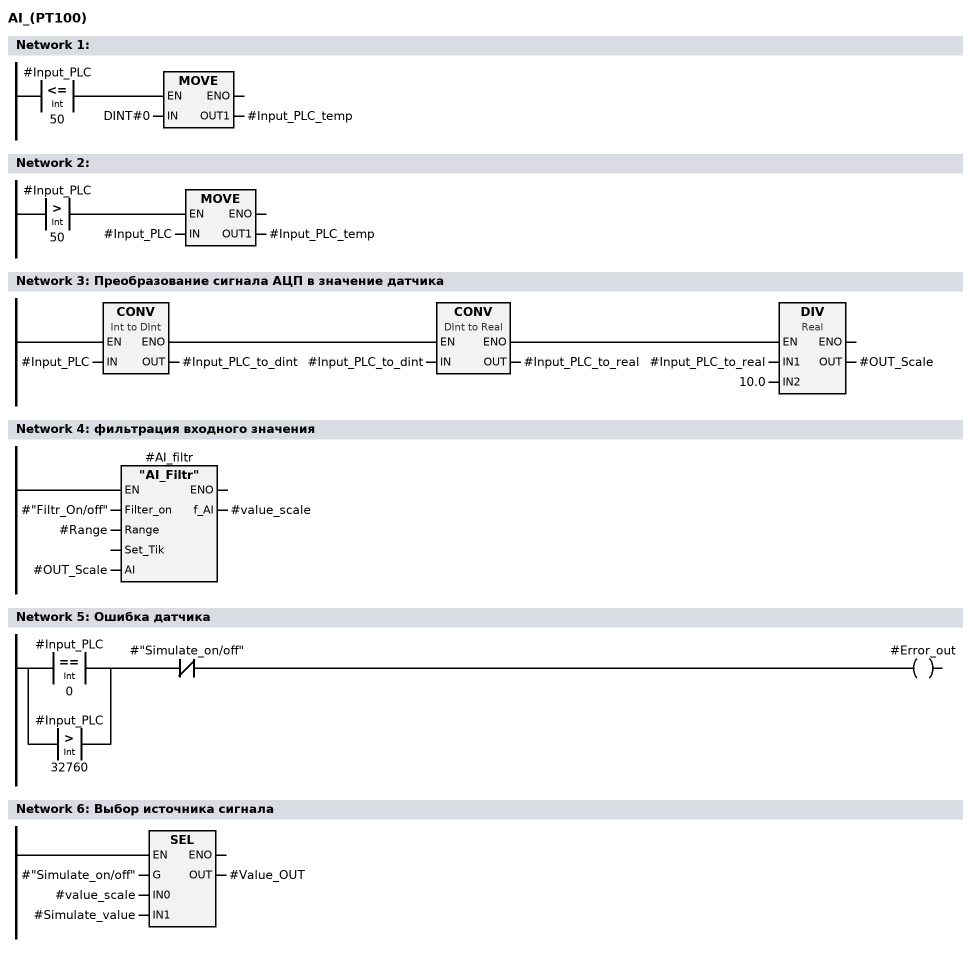
   RUNG wire#powerrail
      { S7_Templates := "SrcType := Int" } LE_Contact(in1 := #Input_PLC, in2 := 50)
      { S7_GenerateENO := "TRUE" } Move(in := DINT#0, out1 => #Input_PLC_temp)
   END_RUNG
   // the same network as SCL:
   IF #Input_PLC <= 50 THEN #Input_PLC_temp := DINT#0; END_IF;
END_REGION

REGION Network 2
   RUNG wire#powerrail
      { S7_Templates := "SrcType := Int" } GT_Contact(in1 := #Input_PLC, in2 := 50)
      { S7_GenerateENO := "TRUE" } Move(in := #Input_PLC, out1 => #Input_PLC_temp)
   END_RUNG
   // the same network as SCL:
   IF #Input_PLC > 50 THEN #Input_PLC_temp := #Input_PLC; END_IF;
END_REGION

REGION Network 3: Преобразование сигнала АЦП в значение датчика
   RUNG wire#powerrail
      { S7_Templates := "[SrcType := Int, DestType := DInt]"; S7_GenerateENO := "TRUE" } Convert(in := #Input_PLC, out => #Input_PLC_to_dint)
      { S7_Templates := "[SrcType := DInt, DestType := Real]"; S7_GenerateENO := "TRUE" } Convert(in := #Input_PLC_to_dint, out => #Input_PLC_to_real)
      { S7_Templates := "SrcType := Real"; S7_GenerateENO := "TRUE" } Div(in1 := #Input_PLC_to_real, in2 := 10.0, out => #OUT_Scale)
   END_RUNG
   // the same network as SCL:
   // ENO of a box is taken as its EN; it also drops when the box reports an error
   #Input_PLC_to_dint := INT_TO_DINT(#Input_PLC);
   #Input_PLC_to_real := DINT_TO_REAL(#Input_PLC_to_dint);
   #OUT_Scale := #Input_PLC_to_real / 10.0;
END_REGION

REGION Network 4: фильтрация входного значения
   RUNG wire#powerrail
      #AI_filtr(Filter_on := #"Filtr_On/off", Range := #Range, Set_Tik :=, AI := #OUT_Scale, f_AI => #value_scale)
   END_RUNG
   // the same network as SCL:
   #AI_filtr(Filter_on := #"Filtr_On/off", Range := #Range, AI := #OUT_Scale, f_AI => #value_scale);   // "AI_Filtr"
END_REGION

REGION Network 5: Ошибка датчика
   RUNG wire#powerrail
      { S7_Templates := "SrcType := Int" } EQ_Contact(in1 := #Input_PLC, in2 := 0)
      wire#w1
      I_Contact( #"Simulate_on/off" )
      Coil( #Error_out )
   END_RUNG
   RUNG wire#powerrail
      { S7_Templates := "SrcType := Int" } GT_Contact(in1 := #Input_PLC, in2 := 32760)
   END_RUNG wire#w1
   // the same network as SCL:
   #Error_out := ((#Input_PLC = 0) OR (#Input_PLC > 32760)) AND NOT #"Simulate_on/off";
END_REGION

REGION Network 6: Выбор источника сигнала
   #Value_OUT := SEL(G := #"Simulate_on/off", IN0 := #value_scale, IN1 := #Simulate_value);
END_REGION
END_FUNCTION_BLOCK

// folder: AI_Signal/Funktion

FUNCTION_BLOCK "AI_Filtr"   // FB14, SCL
{ S7_Optimized_Access := 'FALSE' }
VERSION : 0.1
   VAR_INPUT
      Filter_on : Bool;   // Вкл фильтрации
      Range : Int := 10;   // Кол-во входных значений для вычисления среднего
      Set_Tik : Int := 2;   // Задача периода фильтрации от 1(мин) до 8
      AI : Real;   // Вход значения датчика
   END_VAR
   VAR_OUTPUT
      f_AI : Real;   // выход значения с фильтром или без
   END_VAR
   VAR
      CTU : CTU_INT;   // счетчик для подсчета кол-во вх значений
      Tik : Bool;   // Время фильтрации
      ai_array : Array[0..#Max_Array] of Real;   // Массив значений датчика
      i : Int;   // для цикла ФОР
      sum_AI : Real;   // Суммирование значений с входа датчика
      Avarage_AI : Real;   // Среднее значение датчика
      fRS_set : Bool;   // Для RS тригера
      fRS_res : Bool;   // Для RS тригера
      fRS_out : Bool;   // Для RS тригера
      FullFiltr : Bool;   // Ожидание наполнения значений для вычисления средней
      Res_count : Bool;   // сброс счетчика
   END_VAR
   VAR CONSTANT
      Max_Array : Int := 30;   // Размер массива
   END_VAR
BEGIN

   CASE #Set_Tik OF                   
       1:  
           #Tik := "Time_0.1s";
       2:  
           #Tik := "Time_0.2s";
       3:
           #Tik := "Time_0.4s";
       4:
           #Tik := "Time_0.5s";
       5:
           #Tik := "Time_0.8s";
       6:
           #Tik := "Time_1s";
       7:
           #Tik := "Time_1.6s";
       8:
           #Tik := "Time_2s";
       0:
           #Tik := "Time_0.1s";

       ELSE  
           #Set_Tik := 8;
   END_CASE;  // Выбор периода фильтрации входного сигнала
   REGION RS триггер
       IF #fRS_set THEN
           #fRS_out := true;
       ELSIF #fRS_res AND NOT #fRS_set THEN
           #fRS_out := false;
       END_IF;
   END_REGION

   REGION Подсчет среднего значения входа
       // Statement section REGION
           #CTU(CU := #Tik,
                PV := #Range,
                R := #Res_count,
                Q => #Res_count);                                      // Счетчик для набора значений с входа
           #ai_array[#CTU.CV] := #AI;                                  // Запись значений с входа в массив

           IF #Res_count THEN                                              // СБРОС как счетчик переполниться Для корректной работы счетчика
               #i := 0;
               #sum_AI := 0;
           END_IF;

           IF #Range <> #i THEN                                    // выход из цикла FOR при суммировании всех значений, почему то сам не прекращел подсчет при окончании цикла все время суммировался 
               FOR #i := 0 TO (#Range - 1) DO
                   #sum_AI := #ai_array[#i] + #sum_AI;             // суммирование значений
               END_FOR;
           END_IF;

       #Avarage_AI := #sum_AI / #Range;                             // Вычисление среднего значения
       #fRS_res := NOT #Filter_on;

   END_REGION

   REGION Выбор выхода прямое или фильтрованное значение
       IF #Filter_on THEN                                          //Включение выключение фильтрации
           #fRS_set := #CTU.QD;                                    //При включении фильтра ждем наполнения значениями с входа, пока ждем - отправляем на выход прямое значение входа, далее фильтруем
            #FullFiltr := #fRS_out;

          IF #FullFiltr THEN                                       //Когда фильтр наполнился - вывыодим среднее значение входа
               #f_AI := #Avarage_AI;                              // ЗАпись значения на выход AI
          ELSE
               #f_AI := #AI;                                     // Прямой вывод значения, пока значения не наполнились данными
          END_IF;
       ELSE
           #f_AI := #AI;                                        // Если фильтр выключен, на выход прямое значение с входа
       END_IF; 

   END_REGION
END_FUNCTION_BLOCK

FUNCTION "Calculate_AI" : Void   // FC7, SCL
{ S7_Optimized_Access := 'FALSE' }
VERSION : 0.1
   VAR_INPUT
      IN_sensors : Int;
      Current_max : Real;
      Current_min : Real;
      Code_HL : Real;
      Code_LL : Real;
      Param_Sensor_HL : Real;   // Параметры датчика по паспорту (макс значение)bar, C, итд
      Param_Sensor_LL : Real;   // Параметры датчика по паспорту (мин значение)bar, C, итд
   END_VAR
   VAR_OUTPUT
      signal_Electric : Real;   // выход в электрических ед измерения
      Value_Sensor : Real;   // выход реального значения датчика в ед измерения
   END_VAR
   VAR_TEMP
      sensor_to_real : Real;   // Для конвертации INT to Real
      result_to_out_signal : Real;   // Для вычитания реального значения показания датчика
   END_VAR
BEGIN
       //Convert int to real
   #sensor_to_real := INT_TO_REAL(#IN_sensors);

       // Расчет значения АЦП контроллера в значение эл. ед измерения (I, U) в зависимости от значений на входе
   #signal_Electric := ((#sensor_to_real - #Code_LL) * (#Current_max - #Current_min) / (#Code_HL - #Code_LL))+ #Current_min;
   #result_to_out_signal := #signal_Electric;

   // Расчет значения в реальных единицах измерения датчика (bar, C,) в зависимости от введеных параметров датчика Param_Sensor min/max
   #Value_Sensor := (#result_to_out_signal - #Current_min) * (#Param_Sensor_HL - #Param_Sensor_LL) / (#Current_max - #Current_min) + #Param_Sensor_LL;
END_FUNCTION

// folder: DI_signal

FUNCTION_BLOCK "FB_DI"   // FB15, LAD
TITLE = Блок обработки дискретных входов
{ S7_Optimized_Access := 'FALSE' }
VERSION : 0.1
   VAR_INPUT
      input_value : Bool;   // Входной тэг контроллера
   END_VAR
   VAR_OUTPUT
      Value : Bool;   // Обработанный сигнал
   END_VAR
   VAR_IN_OUT
      stParamDI : "Tipe_DI";
   END_VAR
   VAR
      Time_Delay : Time;   // Время фильтрации для таймера
      Time_On : TON_TIME;   // Фильтр на Вкл
      Time_Off : TON_TIME;   // Фильтр на Выкл
      Nul_Time : Time := T#1MS;   // Откл фильтрации (0)
      bOut_Value : Bool;
   END_VAR
BEGIN

REGION Network 1: Включение фильтрации
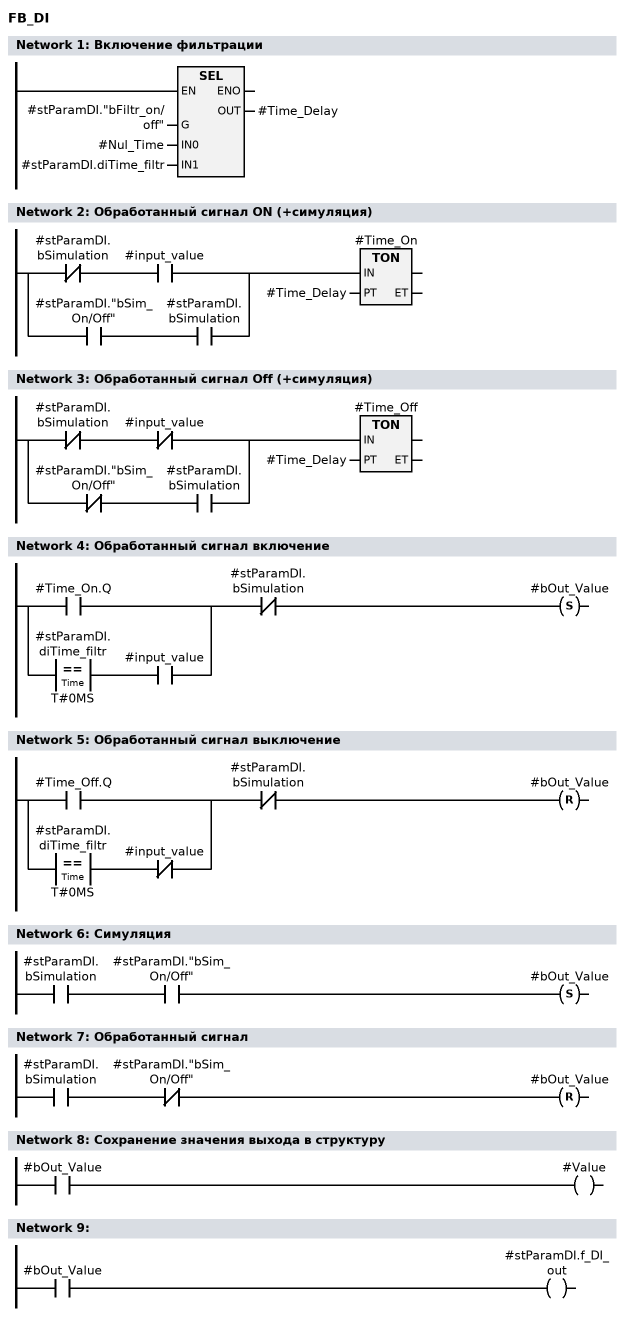
   #Time_Delay := SEL(G := #stParamDI."bFiltr_on/off", IN0 := #Nul_Time, IN1 := #stParamDI.diTime_filtr);
END_REGION

REGION Network 2: Обработанный сигнал ON (+симуляция)
   #Time_On(IN := (NOT #stParamDI.bSimulation AND #input_value) OR (#stParamDI."bSim_On/Off" AND #stParamDI.bSimulation),   // TON
            PT := #Time_Delay);
END_REGION

REGION Network 3: Обработанный сигнал Off (+симуляция)
   #Time_Off(IN := (NOT #stParamDI.bSimulation AND NOT #input_value) OR (NOT #stParamDI."bSim_On/Off" AND #stParamDI.bSimulation),   // TON
             PT := #Time_Delay);
END_REGION

REGION Network 4: Обработанный сигнал включение
   RUNG wire#powerrail
      Contact( #Time_On.Q )
      wire#w1
      I_Contact( #stParamDI.bSimulation )
      S_Coil( #bOut_Value )
   END_RUNG
   RUNG wire#powerrail
      { S7_Templates := "SrcType := Time" } EQ_Contact(in1 := #stParamDI.diTime_filtr, in2 := T#0MS)
      Contact( #input_value )
   END_RUNG wire#w1
   // the same network as SCL:
   IF (#Time_On.Q OR ((#stParamDI.diTime_filtr = T#0MS) AND #input_value)) AND NOT #stParamDI.bSimulation THEN
       #bOut_Value := TRUE;
   END_IF;
END_REGION

REGION Network 5: Обработанный сигнал выключение
   RUNG wire#powerrail
      Contact( #Time_Off.Q )
      wire#w1
      I_Contact( #stParamDI.bSimulation )
      R_Coil( #bOut_Value )
   END_RUNG
   RUNG wire#powerrail
      { S7_Templates := "SrcType := Time" } EQ_Contact(in1 := #stParamDI.diTime_filtr, in2 := T#0MS)
      I_Contact( #input_value )
   END_RUNG wire#w1
   // the same network as SCL:
   IF (#Time_Off.Q OR ((#stParamDI.diTime_filtr = T#0MS) AND NOT #input_value)) AND NOT #stParamDI.bSimulation THEN
       #bOut_Value := FALSE;
   END_IF;
END_REGION

REGION Network 6: Симуляция
   RUNG wire#powerrail
      Contact( #stParamDI.bSimulation )
      Contact( #stParamDI."bSim_On/Off" )
      S_Coil( #bOut_Value )
   END_RUNG
   // the same network as SCL:
   IF #stParamDI.bSimulation AND #stParamDI."bSim_On/Off" THEN #bOut_Value := TRUE; END_IF;
END_REGION

REGION Network 7: Обработанный сигнал
   RUNG wire#powerrail
      Contact( #stParamDI.bSimulation )
      I_Contact( #stParamDI."bSim_On/Off" )
      R_Coil( #bOut_Value )
   END_RUNG
   // the same network as SCL:
   IF #stParamDI.bSimulation AND NOT #stParamDI."bSim_On/Off" THEN #bOut_Value := FALSE; END_IF;
END_REGION

REGION Network 8: Сохранение значения выхода в структуру
   RUNG wire#powerrail
      Contact( #bOut_Value )
      Coil( #Value )
   END_RUNG
   // the same network as SCL:
   #Value := #bOut_Value;
END_REGION

REGION Network 9
   RUNG wire#powerrail
      Contact( #bOut_Value )
      Coil( #stParamDI.f_DI_out )
   END_RUNG
   // the same network as SCL:
   #stParamDI.f_DI_out := #bOut_Value;
END_REGION
END_FUNCTION_BLOCK

// folder: FB - All

FUNCTION_BLOCK "R_trig"   // FB16, SCL
{ S7_Optimized_Access := 'TRUE' }
VERSION : 0.1
   VAR_INPUT
      In : Bool;
   END_VAR
   VAR_OUTPUT
      Q : Bool;
   END_VAR
   VAR
      Click_M : Bool;
   END_VAR
BEGIN
   #Q := #In AND NOT #Click_M;
   #Click_M := #In;
END_FUNCTION_BLOCK

// folder: FB - All/LogickBlocks

FUNCTION_BLOCK "Pump"   // FB1, SCL
{ S7_Optimized_Access := 'FALSE' }
VERSION : 0.1
   VAR_INPUT
      bManualMode : Bool;   // Выбор ручного режима
      bManualStart : Bool;   // Ручной режим - старт
      bManualStop : Bool;   // Ручной режим - стоп
      rManualSpeed : Real;   // Ручной режим - скорость
      bDryRunn : Bool;   // Защита от сухого хода
      bAutoSTop : Bool;   // Остановка насоса
      bAutoStartPerm : Bool;   // Команда на работоу в авто режиме
      rAutoSpeed : Real;   // Скорость в авто режиме
      bАвтоматы : Bool;   // Готовность привода (автоматы)
      bПускатели : Bool;   // Готовность Пускателя
      bDriveRunning : Bool;   // Привод в работе
      bDriveFault : Bool;   // Привод в ошибке
      rMinSpeed : Real;   // Минимальная скорость
      rMaxSpeed : Real := 100.0;   // Максимальная скорость
      bResetFault : Bool;   // Сброс аварии
   END_VAR
   VAR_OUTPUT
      bRunCmd : Bool;   // Пуск частотника
      iSpeedOut : Int;   // Скорость насоса для аналогового выхода
      "rSpeedHMI(0-100)" : Real;   // Скорость работы (0-100) для HMI
      bPumpRunning : Bool;   // Работа
      bPumpFault : Bool;   // Авария
      iStatus : Int;   // Статус (0 - стоп 1 - работа 2 - авария)
   END_VAR
   VAR
      bFaultLatch : Bool;
      bRunRequest : Bool;
      rSpeedPump : Real;   // Скорость насоса
      TON_NotStartRun : TON_TIME;   // ТАймер ожидания сигнала о запуске
      TON_NotContactRun : TON_TIME;   // ТАймер ожидания с контактора
      TON_DryRun : TON_TIME;   // Таймер сухого хода
   END_VAR
BEGIN
   (*
   // 1. Обработка аварий
   // Обработка ожидания сигнала о работе после старта
   IF #bAutoStartPerm THEN
       ;

   END_IF;
   *)

   // 1 Ручной режим
   IF #bManualMode THEN
       // Ручной режим
       IF #bManualStart AND NOT #bManualStop THEN
           #bRunRequest := TRUE;
       ELSIF #bManualStop THEN // OR NOT #bАвтоматы THEN
           #bRunRequest := FALSE;
       END_IF;
   ELSE
       // Автоматический режим
       // 
       //Обработка аварий
       //
       //Таймер ожидания останова по сухому ходу
       #TON_DryRun(IN := NOT #bDryRunn,
                   PT := t#1s);    //
       //--------------------------------------------------------------------------------------------------------
       IF #bAutoStartPerm AND NOT #bAutoSTop AND #bDryRunn THEN
           #TON_NotStartRun(IN := NOT #bDriveRunning AND #bDryRunn, PT := t#5s);  //Таймер ожидания сигнала подтверждения пуска от частотника
           #TON_NotContactRun(IN := NOT #bПускатели, PT := t#10s);  //Таймер ожидания сигнала подтверждения пуска от пускателя


       ELSE
           #TON_NotStartRun(IN :=FALSE,PT := t#5s);
           #TON_NotContactRun(IN := FALSE,PT := t#5s);
       END_IF;
       #bFaultLatch := #TON_NotStartRun.Q OR #TON_NotContactRun.Q OR (#bDriveFault OR NOT #bАвтоматы) OR (NOT #bResetFault AND #bFaultLatch); //Разкоментировать если нужна будет фиксация АЛАРМА, сброс только по входу РЕСЕТ
       #bPumpFault := #bFaultLatch;

       //Старт--------------------------------
       #bRunRequest := #bAutoStartPerm AND NOT #bPumpFault AND NOT #TON_DryRun.Q;
   END_IF;

   // 3. Задание скорости
   IF #bManualMode THEN
       #"rSpeedHMI(0-100)" := LIMIT(MN := #rMinSpeed, IN := #rManualSpeed, MX := #rMaxSpeed);
   ELSE
       #"rSpeedHMI(0-100)" := LIMIT(MN := #rMinSpeed, IN := #rAutoSpeed, MX := #rMaxSpeed);
   END_IF;

   // Преобразование значения от 0-100 до 0-27648 для аналогового выхода
   #iSpeedOut := REAL_TO_INT((#"rSpeedHMI(0-100)"/ 100.0) * 27648.0);

   // 4. Выходные команды и статусы
   // Команды старт
   #bRunCmd := #bRunRequest;

   //Выход статуса для HMI
   #bPumpRunning := #bDriveRunning AND #bRunCmd AND NOT #bAutoSTop OR (#bManualStart AND #bManualMode);



   // 5. Числовой статус (для HMI/SCADA)
   IF #bFaultLatch THEN
       #iStatus := 2; // Авария
   ELSIF #bPumpRunning THEN
       #iStatus := 1; // Работа
   ELSE
       #iStatus := 0; // Стоп
   END_IF;

   IF #bAutoSTop AND NOT #bManualMode THEN
       #bRunCmd := FALSE;
   END_IF;
END_FUNCTION_BLOCK

FUNCTION_BLOCK "FB_GlobalStateManager"   // FB2, SCL
{ S7_Optimized_Access := 'FALSE' }
VERSION : 0.1
   VAR_INPUT
      bStartCmd : Bool;   // Команда на старт от HMI
      bConfirmStart : Bool;   // Подтверждение оператора
      bResetFault : Bool;   // Сброс ошибки
      bAllSetpointsReached : Bool;   // // Все температуры достигли уставок
      bNoFaults : Bool;   // Нет аварий
      tStartTimeout : Time := T#30m;   // Время за которое пастер выходит на режим
      tReadyDelay : Time := t#10s;   // Время ожидания при выходе на режим до готовности
   END_VAR
   VAR_OUTPUT
      eState : Int;   // Текущее состояние
      bConveyorEnable : Bool;   // Разрешение на работу конвейера
      bSystemReady : Bool;   // Готовность системы
      bSystemFault : Bool;   // Состояние Fault
      sStatusText : WString;   // Текст для HMI
   END_VAR
   VAR
      tonStartTimeout : TON_TIME;   // Таймер выхода на режим
      tonReadyDelay : TON_TIME;   // Таймер готовности
   END_VAR
   VAR CONSTANT
      cSTATE_IDLE : Int;
      cSTATE_CHECK : Int := 10;
      cSTATE_STARTING : Int := 20;
      cSTATE_READY_DELAY : Int := 30;
      cSTATE_READY : Int := 40;
      cSTATE_FAULT : Int := 99;
      sText1 : String := 'Waiting';
   END_VAR
BEGIN
   // Сброс таймеров при неактивных состояниях (по требованию 1)
   IF #eState <> #cSTATE_STARTING THEN
       #tonStartTimeout(IN := FALSE,
                        PT := #tStartTimeout);
   END_IF;

   IF #eState <> #cSTATE_READY_DELAY THEN
       #tonReadyDelay(IN := FALSE,
                      PT := #tReadyDelay);
   END_IF;

   // Глобальная проверка аварии (по требованию 4)
   IF NOT #bNoFaults AND #eState <> #cSTATE_FAULT THEN
       #eState := #cSTATE_FAULT;
       #bSystemFault := TRUE;
       #bConveyorEnable := FALSE; // Принудительный останов (по требованию 2)
   ELSIF NOT #bStartCmd THEN
       #eState := #cSTATE_IDLE;
   END_IF;


   REGION Основная логика

       // Основной CASE
       CASE #eState OF
           #cSTATE_IDLE:
               #bConveyorEnable := FALSE;
               IF #bStartCmd AND #bNoFaults THEN // Запрет старта при аварии
                   #eState := #cSTATE_CHECK;
               END_IF;

           #cSTATE_CHECK:
               // Проверка уже в глобальном условии, дублирование не нужно
               #eState := #cSTATE_STARTING;

           #cSTATE_STARTING:
               IF #bAllSetpointsReached THEN
                   #eState := #cSTATE_READY_DELAY;
               ELSIF #tonStartTimeout.Q THEN
                   #eState := #cSTATE_FAULT;
               END_IF;

           #cSTATE_READY_DELAY:
               IF #tonReadyDelay.Q THEN
                   #eState := #cSTATE_READY;
               END_IF;

           #cSTATE_READY:
               #bSystemReady := TRUE;
               IF #bConfirmStart THEN
                   #bConveyorEnable := TRUE;
               END_IF;

           #cSTATE_FAULT:
               #bSystemFault := TRUE;
               #bConveyorEnable := FALSE; // Гарантированный останов
               IF #bResetFault AND #bNoFaults THEN
                   #eState := #cSTATE_IDLE;
                   #bSystemFault := FALSE;
               END_IF;

           ELSE
               #eState := #cSTATE_IDLE;
       END_CASE;

   END_REGION


   // Обновление таймеров (после логики состояний!)
   #tonStartTimeout(IN := (#eState = #cSTATE_STARTING) AND NOT #bAllSetpointsReached,
                    PT := #tStartTimeout);
   #tonReadyDelay(IN := (#eState = #cSTATE_READY_DELAY),
                  PT := #tReadyDelay);
END_FUNCTION_BLOCK

FUNCTION_BLOCK "Valve(c/o)"   // FB3, SCL
{ S7_Optimized_Access := 'FALSE' }
VERSION : 0.1
   VAR_INPUT
      bAuto_OpenCmd : Bool;   // Команда открыть (автомат)
      bManualMode : Bool;   // Ручной режим (TRUE)
      bManualOpen : Bool;   // Команда открыть в ручном режиме
      bFeedbackOpen : Bool;   // Обратная связь "Открыт"
      tMaxTime : Time;   // Время на открытие
      bResetAlarm : Bool;   // Сброс аварии
      bHaveFeedback : Bool;   // Есть ли обратная связь (0 - нет, 1 есть)
   END_VAR
   VAR_OUTPUT
      bValveOpen : Bool;   // Управляющий выход
      iValveState : Int;   // 0 = Закрыт, 1 = Открыт, 2 = Авария
      bValveFault : Bool;   // Авария
   END_VAR
   VAR
      tiOpenTimer : TON_TIME;   // Таймер на открытие
      bWaitingOpen : Bool;   // Флаг ожидания открытия
      bEnableTimer : Bool;   // Флаг активации таймера
   END_VAR
BEGIN

   // Обновление таймера — всегда в одном месте, вне условий
   #tiOpenTimer(
                IN := #bEnableTimer,
                PT := #tMaxTime
   );

   // Сброс
   IF #bResetAlarm THEN
       #bValveFault := FALSE;
       #bWaitingOpen := FALSE;
       #bEnableTimer := FALSE;
   END_IF;

   // === Режим: РУЧНОЙ ===
   IF #bManualMode THEN
       #bValveOpen := #bManualOpen;
       #bValveFault := FALSE;          // Аварии в ручном режиме не учитываются
       #bEnableTimer := FALSE;
       #bWaitingOpen := FALSE;

       // === Режим: АВТО ===
   ELSE

           // Управление выходом с учетом аварии, с контролем обратной связи
        IF #bAuto_OpenCmd AND NOT #bValveFault THEN
                   #bValveOpen := TRUE;
        ELSE
                   #bValveOpen := FALSE;
               END_IF;

               //  Проверяем, есть ли контроль обратной связи
        IF #bHaveFeedback THEN
            // Контроль открытия
            IF #bAuto_OpenCmd AND NOT #bFeedbackOpen AND NOT #bValveFault THEN
                #bEnableTimer := TRUE;
                #bWaitingOpen := TRUE;
            ELSE
                #bEnableTimer := FALSE;
                ;
                IF #bFeedbackOpen THEN
                    #bWaitingOpen := FALSE;
                END_IF;
            END_IF;
        END_IF;


           // Авария
           IF #tiOpenTimer.Q AND #bWaitingOpen THEN
               #bValveFault := TRUE;
               #bWaitingOpen := FALSE;
           END_IF;

   END_IF;


   // Состояние клапана
   IF #bValveFault THEN
       #iValveState := 2;       // Авария
   ELSIF #bHaveFeedback AND #bFeedbackOpen  THEN
       #iValveState := 1;       // Открыт
   ELSIF NOT #bHaveFeedback AND (NOT #bManualMode AND #bAuto_OpenCmd) OR (#bManualOpen AND #bManualMode) THEN
       #iValveState := 1;       // Открыт 
   ELSE
       #iValveState := 0;       // Закрыт
   END_IF;
END_FUNCTION_BLOCK

FUNCTION_BLOCK "Valve(regul)"   // FB4, SCL
{ S7_Optimized_Access := 'FALSE' }
VERSION : 0.1
   VAR_INPUT
      bManualMode : Bool;   // TRUE = ручной режим, FALSE = автоматический режим
      rAutoSetpoint : Real;   // Уставка открытия клапана в % (0.0–100.0) в автомате
      "bAutoOpen/Close" : Bool;   // Выход Do в автоматическом режиме
      rManualSetpoint : Real;   // Уставка открытия клапана в % (0.0–100.0) в ручном режиме
      "bManualOpen/Close" : Bool;   // Управление выходом открыть/закрыть
   END_VAR
   VAR_OUTPUT
      iAnalogOutput : Int;   // Значение для аналогового выхода (0–27648)
      rValvePosPercent : Real;   // Текущее % открытия клапана для HMI
      bStatusValveOpen : Int;   // Статус сигнал "клапан открыт" (TRUE, если >0%)
      "bOut_Open/Close" : Bool;   // выход для открытия клапана
   END_VAR
   VAR
      rSetpointPercent : Real;   // Расчётная уставка % открытия в текущем режиме
   END_VAR
BEGIN
       // Выбор уставки в зависимости от режима
       IF #bManualMode THEN
           #rSetpointPercent := #rManualSetpoint;
           #"bOut_Open/Close" := #"bManualOpen/Close";
       ELSE
           #rSetpointPercent := #rAutoSetpoint;
           #"bOut_Open/Close" := #"bAutoOpen/Close";
       END_IF;

       // Ограничение % от 0.0 до 100.0
       IF #rSetpointPercent < 0.0 THEN
           #rSetpointPercent := 0.0;
       ELSIF #rSetpointPercent > 100.0 THEN
           #rSetpointPercent := 100.0;
       END_IF;

       // Перевод % в значение для аналогового выхода
       #iAnalogOutput := REAL_TO_INT((#rSetpointPercent / 100.0) * 27648.0);

           // Вывод значения для HMI
       #rValvePosPercent := #rSetpointPercent;

       // Статус клапана для Панели HMI
       IF #rSetpointPercent > 0.0 AND #"bOut_Open/Close" THEN
           #bStatusValveOpen := 1;
       ELSE
           #bStatusValveOpen := 0;
       END_IF;
       ;
END_FUNCTION_BLOCK

FUNCTION_BLOCK "FB_Управление конвейером"   // FB5, SCL
{ S7_Optimized_Access := 'FALSE' }
VERSION : 0.1
   VAR_INPUT
      bEnable : Bool;   // Общий флаг работы системы
      bStartCmd : Bool;   // Команда на запуск от HMI, по кнопке из окна подтверждения
      bAllZonesInSetpoint : Bool;   // Все зоны достигли уставок
      bGlobalFault : Bool;   // Авария по системе
      bZoneHasPriority : Bool;   // У зоны с отклонением есть приоритет
      dwDeltaTempDelayMin : DWord;   // Задержка (мин), прежде чем остановить конвейер при отклонении
      dwResumeDelayMin : DInt;   // Время возврата после нормализации
   END_VAR
   VAR_OUTPUT
      bConveyorRun : Bool;   // Команда на пуск частотников
      bReadyToStart : Bool;   // Готовность к работе конвейера
      bWaitingConfirm : Bool;   // Ждём подтверждения от оператора, вывод окна на HMI
      bPaused : Bool;   // Конвейер остановлен по отклонению
   END_VAR
   VAR
      bStarted : Bool;   // Внутреннее состояние — процесс стартовал
      tiPauseTimer : TON_TIME;   // Таймер задержки перед остановкой
      tiResumeTimer : TON_TIME;   // Таймер ожидания перед возобновлением
      aZoneS_Status : Array[1..5] of "ZoneStatus";   // Массив для сбора состояния зон
      i : Int;
   END_VAR
   // tiPauseTimer.PT := T#1s;
   // tiResumeTimer.PT := T#1s;
BEGIN

   // Проверка на наличие флага обей работы системы
   IF NOT #bEnable THEN
       #bReadyToStart := FALSE;
       #bWaitingConfirm := FALSE;
       #bConveyorRun := FALSE;
       #bPaused := FALSE;
       #tiPauseTimer.IN := FALSE;
       #tiResumeTimer.IN := FALSE;
       RETURN;
   END_IF;



   // Условия готовности к запуску
   IF NOT #bStarted AND NOT #bGlobalFault AND #bAllZonesInSetpoint THEN
       #bReadyToStart := TRUE;

           // Команда на старт — вручную подтверждена
           IF NOT #bStartCmd THEN
               #bWaitingConfirm := TRUE;
           END_IF;

   ELSE
       #bReadyToStart := FALSE;
       #bWaitingConfirm := FALSE;
   END_IF;



   IF #bStartCmd AND #bReadyToStart THEN
       #bStarted := TRUE;
       #bWaitingConfirm := FALSE;
   END_IF;

   // После старта разрешаем работу, если нет аварий и температур в норме
   IF #bStarted AND NOT #bGlobalFault THEN

       IF NOT #bAllZonesInSetpoint THEN
           IF #bZoneHasPriority THEN
               // Включаем таймер паузы, задержка перед остановкой
               #tiPauseTimer(IN := TRUE,
                             PT := (#dwDeltaTempDelayMin * 60000)) //В минутах
               ;
           ELSE
               #tiPauseTimer(IN := FALSE,PT := t#0s);
           END_IF;

           // Переход в паузу
           IF #tiPauseTimer.Q THEN
               #bPaused := TRUE;
               #bConveyorRun := FALSE;
               #tiResumeTimer(IN := FALSE, PT := t#0s); // Сброс таймера возобновления

           END_IF;

       ELSE
           // Температуры вернулись в норму — запускаем таймер на возврат
           IF #bPaused THEN
               #tiResumeTimer(IN := TRUE,
                              PT := (#dwResumeDelayMin * 60000)) // в минутах
               ;
               // Возвращаемся к работе
               IF #tiResumeTimer.Q THEN
                   #bPaused := FALSE;
                   #bConveyorRun := TRUE;
                   #tiResumeTimer(IN := FALSE, PT := t#0s); // сброс таймера
               END_IF;
           ELSE
               #bConveyorRun := TRUE;
               #tiPauseTimer(IN := FALSE, PT := t#0s); // сброс
               #tiResumeTimer(IN := FALSE,PT := t#0s);
           END_IF;
       END_IF;
   ELSE
       // Если глобальная авария — всё стоп
       #bConveyorRun := FALSE;
       #bPaused := FALSE;
       #bStarted := FALSE;
       #tiPauseTimer(IN := FALSE, PT := t#0s);
       #tiResumeTimer(IN := FALSE,PT := t#0s);
       #bWaitingConfirm := FALSE;
   END_IF;
END_FUNCTION_BLOCK

FUNCTION_BLOCK "FB_Motor_Conveyor"   // FB6, SCL
{ S7_Optimized_Access := 'FALSE' }
VERSION : 0.1
   VAR_INPUT
      bManualMode : Bool;   // Выбор ручного режима
      bManualStart : Bool;   // Ручной режим - старт
      bManualStop : Bool;   // Ручной режим - стоп
      rManualSpeed : Real;   // Ручной режим - скорость
      bAutoStartPerm : Bool;   // Команда на работоу в авто режиме
      rAutoSpeed : Real;   // Скорость в авто режиме
      bDriveReady : Bool;   // Готовность привода (автоматы)
      bDriveRunning : Bool;   // Привод в работе
      bDriveFault : Bool;   // Привод в ошибке
      rMinSpeed : Real;   // Минимальная скорость
      rMaxSpeed : Real;   // Максимальная скорость
      bResetFault : Bool;   // Сброс аварии
   END_VAR
   VAR_OUTPUT
      bRunCmd : Bool;   // Пуск частотника
      "rSpeedHMI(0-100)" : Real;   // Скорость работы (0-100) для HMI
      iSpeedOut : Int;   // Скорость насоса для аналогового выхода
      bPumpRunning : Bool;   // Работа
      bPumpFault : Bool;   // Авария
      iStatus : Int;   // Статус (0 - стоп 1 - работа 2 - авария)
   END_VAR
   VAR
      bFaultLatch : Bool;
      bRunRequest : Bool;
      rSpeedPump : Real;   // Скорость насоса
   END_VAR
BEGIN
   // 1. Обработка аварий
   #bFaultLatch := (#bDriveFault OR #bFaultLatch) AND NOT #bResetFault;
   #bPumpFault := #bFaultLatch;

   // 2. Формирование команды "Пуск"
   IF #bManualMode THEN
       // Ручной режим
       IF #bManualStart AND NOT #bManualStop THEN
           #bRunRequest := TRUE;
       ELSIF #bManualStop OR NOT #bDriveReady THEN
           #bRunRequest := FALSE;
       END_IF;
   ELSE
       // Автоматический режим
       #bRunRequest := #bAutoStartPerm AND NOT #bDriveFault;
   END_IF;

   // 3. Задание скорости
   IF #bManualMode THEN
       #"rSpeedHMI(0-100)" := LIMIT(MN := #rMinSpeed, IN := #rManualSpeed, MX := #rMaxSpeed);
   ELSE
       #"rSpeedHMI(0-100)" := LIMIT(MN := #rMinSpeed, IN := #rAutoSpeed, MX := #rMaxSpeed);
   END_IF;

   // Преобразование значения от 0-100 до 0-27648 для аналогового выхода
   #iSpeedOut := REAL_TO_INT((#"rSpeedHMI(0-100)"/ 100.0) * 27648.0);

   // 4. Выходные команды и статусы
   #bRunCmd := #bRunRequest AND NOT #bFaultLatch AND #bDriveReady;
   #bPumpRunning := #bDriveRunning AND #bRunCmd;

   // 5. Числовой статус (для HMI/SCADA)
   IF #bFaultLatch THEN
       #iStatus := 2; // Авария
   ELSIF #bPumpRunning THEN
       #iStatus := 1; // Работа
   ELSE
       #iStatus := 0; // Стоп
   END_IF;
END_FUNCTION_BLOCK

FUNCTION_BLOCK "FB_Аварии"   // FB7, SCL
{ S7_Optimized_Access := 'FALSE' }
VERSION : 0.1
   VAR_INPUT
      Rtrig_Reset : Bool;
   END_VAR
   VAR_OUTPUT
      ALARM_Active : Bool;   // Флаг активной аварии
   END_VAR
   VAR
      LatchedEmergency : Bool;   // Зафиксированная аварийная ситуация
      bAlarmAvtomats : Bool;   // Авария автоматов
      bAlarmAI : Bool;   // Авария аналоговых датчиков
      bAlarmPumps : Bool;   // Авария насосов
      bAlarmConveyors : Bool;   // Авария Конвейеров
      bAlarmFVs : Bool;   // Авария клапанов
      bAlarmDI_all : Bool;   // Авария по дискретным входам "общая"
      bAlarmLowLevel : Bool;   // Авария по низкому уровню емкостей
      mReset : Bool;
      TON_LowLevel : TON_TIME;   // Таймер для аварийного уровня емкостей
      bResetaALARM : Bool;   // Сброс аварии (кнопка на панели/системе)
   END_VAR
   VAR_TEMP
      nAi : Int;
      nPump : Int;
      nConv : Int;
      nFV : Int;
      nAvtomat : Int;
      numPump : Int;
   END_VAR
BEGIN
   REGION Предварительное отрицание
       // Сброс в 0 при отсутсвии аварий для цикла и массивов
       #bAlarmAvtomats := FALSE;
       #bAlarmAI := FALSE;
       #bAlarmPumps := FALSE;
       #bAlarmConveyors := FALSE;
       #bAlarmFVs := FALSE;


   END_REGION



   //Авария автоматические выключатели
   //--------------------------
   (*
   "Alarms".Avtomat_Off[1].ALARM := NOT "Conveyor".Conveyor_1.bIn_AutomatState;
   "Alarms".Avtomat_Off[2].ALARM := NOT "Conveyor".Conveyor_2.bIn_AutomatState;
   "Alarms".Avtomat_Off[3].ALARM := NOT "Conveyor".Conveyor_3.bIn_AutomatState;
   "Alarms".Avtomat_Off[4].ALARM  :=  NOT "Pumps".Pump_1.bIn_AutomatState;
   "Alarms".Avtomat_Off[5].ALARM  :=  NOT "Pumps".Pump_2.bIn_AutomatState;
   "Alarms".Avtomat_Off[6].ALARM  :=  NOT "Pumps".Pump_3.bIn_AutomatState;
   "Alarms".Avtomat_Off[7].ALARM  :=  NOT "Pumps".Pump_4.bIn_AutomatState;
   "Alarms".Avtomat_Off[8].ALARM  :=  NOT "Pumps".Pump_5.bIn_AutomatState;
   "Alarms".Avtomat_Off[9].ALARM  :=  NOT "Pumps".Pump_6.bIn_AutomatState;
   "Alarms".Avtomat_Off[10].ALARM  :=  NOT "Pumps".Pump_7.bIn_AutomatState;
   "Alarms".Avtomat_Off[11].ALARM  :=  NOT "Vent".Vent_1.bIn_AutomatState;


   FOR #nAvtomat := 1 TO 11 DO
       IF "Alarms".Avtomat_Off[#nAvtomat].ALARM THEN
           #bAlarmAvtomats := TRUE;
       END_IF;
   END_FOR;
   *)
   //Авария аналоговых входов
   //--------------------------
   FOR #nAi := 1 TO 7 DO
       IF "Alarms".Ai_Alarm[#nAi].ALARM THEN
           #bAlarmAI := TRUE;
       END_IF;
   END_FOR;

   //Авария НАСОСОВ
   //--------------------------

   FOR #nPump := 1 TO 7 DO
       IF "Alarms".Pump_Alarm[#nPump].ALARM THEN
           #bAlarmPumps := TRUE;
           #numPump := #nPump;

       END_IF;
   END_FOR;

   //Авария КОНВЕЙЕРОВ
   //--------------------------

   FOR #nConv := 1 TO 4 DO
       IF "Alarms".Conveyor_Alarm[#nConv].ALARM THEN
           #bAlarmConveyors := TRUE;
       END_IF;
   END_FOR;

   //Авария Клапанов
   //--------------------------

   FOR #nFV := 1 TO 7 DO
       IF "Alarms".FV_Alarm[#nFV].ALARM THEN
           #bAlarmFVs := TRUE;
       END_IF;
   END_FOR;

   //Авария под давлению
   //--------------------------
   "AlarmPress" := "Control_Press_DB".PressWater.bAlarm_Press OR "Control_Press_DB".PressSteam.bAlarm_Press OR "Control_Press_DB".PressGlikol.bAlarm_Press;

   //Авария по нижним датчикам уровня емкостей
   //

   //#bAlarmLowLevel := NOT "My_VarS".b_Woter_LowLevel_T1;

   //Авария по входам DI
   //---------------------------

   #bAlarmDI_all :="Alarms"."xE-Stop_1" OR
                   "Alarms"."xE-Stop_2" OR
                   "Alarms"."xE-Stop_3" OR
                   "Alarms".xVoltRele OR
                   "Alarms".xSensorConveyorZator_1 OR
                  // "Alarms".xSensorConveyorZator_2 OR
                   "Alarms".xLongPauseConv OR
                   "Alarms".xLongWaitZoneOk;

   //Обработка всех аварий с выводом сигнала наличия АВАРИЯ
   //----------------------------------------------------------------
                   IF #bAlarmAvtomats OR
                       #bAlarmAI OR
                       #bAlarmPumps OR
                       #bAlarmConveyors OR
                       #bAlarmFVs OR
                       #bAlarmDI_all OR
                       #bAlarmLowLevel
                   THEN

                       #ALARM_Active := TRUE;
                   END_IF;
     (*                     
   //Отлавливаем фронт Ресета....................................

   #bResetaALARM := #Rtrig_Reset AND NOT #mReset;
   #mReset := #Rtrig_Reset;
   *)

    //Если нужен жесткий сбро, игнорирует все аварии                      
   #bResetaALARM := #Rtrig_Reset;

   //-------------------------------------------------------------                       
                          // Сброс аварии
   IF #bResetaALARM THEN
       #ALARM_Active := FALSE;
   END_IF;
END_FUNCTION_BLOCK

FUNCTION_BLOCK "FB_Zone_Control"   // FB8, SCL
{ S7_Optimized_Access := 'FALSE' }
VERSION : 0.1
   VAR_INPUT
      bNewStart : Bool;   // Обнаружение нового старта, уставка без дельты
      rTempActual : Real;   // Температура с датчика
      rTempSetpoint : Real;   // Уставка температуры
      rDeltaDown : Real;   // Верхнее Допустимое отклонение от уставки
      rDeltaUp : Real;   // Верхнее Допустимое отклонение от уставки
      bPriority : Bool;   // Приоритет управления конвейером (1 - стоп конвейер)
   END_VAR
   VAR_OUTPUT
      ZoneStatusOut : "ZoneStatus";
      bInSetpoint : Bool;
      bOutOfRange : Bool;
      bHasPriority : Bool;
   END_VAR
   VAR
      R_Trig_Start : "R_trig";
      "#bNewStartCLic" : Bool;
      bSetpointReachedOnce : Bool;
   END_VAR
BEGIN
   // --- Сброс флага при необходимости ---
   // 
       //----Отслеживание нажания старта, по верхнему фронту-----
   #R_Trig_Start("In":= #bNewStart,Q => #"#bNewStartCLic");

   IF #"#bNewStartCLic" THEN
       #bSetpointReachedOnce := FALSE;
   END_IF;

   // --- Фиксация первого достижения уставки (точно или ±0.1) ---
   IF NOT #bSetpointReachedOnce AND ABS(#rTempActual - #rTempSetpoint) <= 1 THEN
       #bSetpointReachedOnce := TRUE;
   END_IF;

   // --- Расчёт попадания в уставку с учетом асимметричной дельты ---
   IF #bSetpointReachedOnce THEN
       #ZoneStatusOut.bInSetpoint := (#rTempActual >= (#rTempSetpoint - #rDeltaDown)) AND
                                       (#rTempActual <= (#rTempSetpoint + #rDeltaUp));
   ELSE
       // До первого достижения — строгое приближение (или узкая дельта)
       #ZoneStatusOut.bInSetpoint := ABS(#rTempActual - #rTempSetpoint) <= 1;
   END_IF;

   //Контроль зоны выхода из уставок значительно, греем снова до уставки до разрешения на старт

   IF (#rTempActual < (#rTempSetpoint - #rDeltaDown)) OR
       (#rTempActual > (#rTempSetpoint + #rDeltaUp)) THEN
       #bSetpointReachedOnce := FALSE;
   END_IF;


   // --- Остальные сигналы ---
   #ZoneStatusOut.bOutOfRange := NOT #ZoneStatusOut.bInSetpoint;
   #ZoneStatusOut.bHasPriority := #bPriority;

   // Зеркалируем, если нужно
   #bInSetpoint := #ZoneStatusOut.bInSetpoint;
   #bOutOfRange := #ZoneStatusOut.bOutOfRange;
   #bHasPriority := #ZoneStatusOut.bHasPriority;
END_FUNCTION_BLOCK

FUNCTION_BLOCK "FB_check_For_Start"   // FB9, SCL
{ S7_Optimized_Access := 'FALSE' }
VERSION : 0.1
   VAR_INPUT
      xHMI_Start : Bool;   // кнопка старта с HMI
      xEmergency_Stop : Bool;   // аварийный стоп
      xSystem_Ready : Bool;   // Готовность всех систем
      xStopHMI : Bool;   // Кнопка СТОП на HMI
   END_VAR
   VAR_OUTPUT
      xStart_Allowed : Bool;   // Разрешение на РАБОТУ
      xStart : Bool;   // Работа пастеризатора
   END_VAR
   VAR
      "m" : Bool;   // memory
   END_VAR
BEGIN

   //Проверка на разрешение работы.
   //
   IF NOT #xEmergency_Stop AND #xSystem_Ready THEN
       #xStart_Allowed := TRUE;
   ELSE
       #xStart_Allowed := FALSE;
   END_IF;

   #xStart := (#xStart OR #xHMI_Start) AND NOT (#xEmergency_Stop OR #xStopHMI);
END_FUNCTION_BLOCK

FUNCTION_BLOCK "FB_Stiril_CheckZoneStatus"   // FB10, SCL
{ S7_Optimized_Access := 'FALSE' }
VERSION : 0.1
   VAR_OUTPUT
      bAllZones_Redy : Bool;   // Выход состояния всех зон ОК
      bPriority_Stop : Bool;   // Выход 1 - если есть метка остановки конвейера
      iZonesNumberFail : Int;   // ВЫход с Номером зоны
   END_VAR
   VAR
      aZoneS_Status : Array[1..10] of "ZoneStatus";   // Массив с данными по всем зонам
      i : Int;
      AllZone_Ok : Bool;   // Состояние всех зон ОК
      HaveStopPriority : Bool;   // В зоне есть метка для остановки конвейера
      iNumber : Int;   // Номер зоны, где отклонение температуры
   END_VAR
BEGIN

   //Что бы не контролировал готовность зоны 4 ее не надо контролировать
   //"ЗОНЫ_Параметры".Zone_4.bOUT_ZoneStatus.bInSetpoint := TRUE;
   //-------------------------------------------------------------------------------------------//
   //
           // ----Сбор данных по всем зонам в массив для обработки-----
           #aZoneS_Status[1] := "Зоны_Стерилизации_Парам"."Steril_Zona-1".bOUT_ZoneStatus;
           #aZoneS_Status[2] := "Зоны_Стерилизации_Парам"."Steril_Zona-2".bOUT_ZoneStatus;
           #aZoneS_Status[3] := "Зоны_Стерилизации_Парам"."Steril_Zona-3".bOUT_ZoneStatus;
           #aZoneS_Status[4] := "Зоны_Стерилизации_Парам"."Steril_Zona-4".bOUT_ZoneStatus;
           #aZoneS_Status[5] := "Зоны_Стерилизации_Парам"."Steril_Zona-5".bOUT_ZoneStatus;
           #aZoneS_Status[6] := "Зоны_Стерилизации_Парам"."Steril_Zona-6".bOUT_ZoneStatus;
           #aZoneS_Status[7] := "Зоны_Стерилизации_Парам"."Steril_Zona-7".bOUT_ZoneStatus;
           #aZoneS_Status[8] := "Зоны_Стерилизации_Парам"."Steril_Zona-8".bOUT_ZoneStatus;
           #aZoneS_Status[9] := "Зоны_Стерилизации_Парам"."Steril_Zona-9".bOUT_ZoneStatus;
           #aZoneS_Status[10] := "Зоны_Стерилизации_Парам"."Steril_Zona-10".bOUT_ZoneStatus;


           //Сброс маркеров по умолчанию----
   #AllZone_Ok := TRUE;    
   #HaveStopPriority := FALSE;
   #iNumber := 0;
              // ----Цикл для перебора всех зон значение выставить по количеству зон----
   FOR #i := 1 TO 10 DO
       IF NOT #aZoneS_Status[#i].bInSetpoint THEN
           #AllZone_Ok := FALSE;
           #iNumber := #i;
           IF #aZoneS_Status[#i].bHasPriority THEN
               #HaveStopPriority := TRUE;
           END_IF;
       END_IF;
   END_FOR;

   /// Присвоение переменных к выходам
   #bAllZones_Redy := #AllZone_Ok;
   #bPriority_Stop := #HaveStopPriority;
   #iZonesNumberFail := #iNumber;
END_FUNCTION_BLOCK

FUNCTION_BLOCK "FB_ПЕ_Control"   // FB11, SCL
{ S7_Optimized_Access := 'TRUE' }
VERSION : 0.1
   VAR_INPUT
      bRunRequest : Bool;   // Запрос на работу
      rSpeedPercent : Real;   // Заданная скорость от оператора (0…100%)
      rPESetpoint : Real;   // Заданное количество ПЕ
      rConveyorLength : Real := 8.3;   // Длина зоны выдержки, м
      rVmax : Real := 0.0085;   // Макс скорость м/мин
      rZParam : Real := 1.393;   // Коэффициент z (1.393 обычно)
      rTref : Real := 60.0;   // Базовая температура (обычно 60°C)
      rTmin : Real;   // Мин допустимая температура
      rTmax : Real := 75.0;   // Макс допустимая температура
      bManualMode : Bool;   // Режим "ручной расчёт температуры"
      rManualTemp : Real;   // Температура в ручном режиме
      tStopTolerance : Time;   // Допустимое время простоя
   END_VAR
   VAR_OUTPUT
      rTempSetpoint : Real;   // Уставка температуры
      rHoldTime : Real;   // Время выдержки в мин
      rConveyorSpeed : Real;   // Скорость конвейера (м/мин)
      rPENeededPerMin : Real;   // Требуемое ПЕ в минуту
      bTempValid : Bool;   // Температура в пределах допустимого
      bAlarmTempHigh : Bool;   // Температура превышает максимум
      bAlarmTempLow : Bool;   // Температура ниже минимума
      bStoppedTooLong : Bool;   // Превышено время простоя
      bAlarmTempOverride : Bool;   // Принудительная уставка из-за аварии
   END_VAR
   VAR RETAIN
      rSpeedRatio : Real;   // Отношение скорости
      rLogArg : Real;   // Аргумент логарифма
   END_VAR
   VAR
      TON_StopDelay : TON_TIME;   // Таймер задержки останова
   END_VAR
BEGIN
   // Блок управления уставкой температуры по ПЕ и скорости
   // Сначала сброс в случае остановки
   IF NOT #bRunRequest THEN
       //#rTempSetpoint := 0.0;
       #rHoldTime := 0.0;
       #rConveyorSpeed := 0.000;
       #bTempValid := TRUE;
       #bAlarmTempHigh:= FALSE;
       #bAlarmTempLow := FALSE;
       #bAlarmTempOverride := FALSE;
       #bStoppedTooLong := FALSE;
       #TON_StopDelay(IN := FALSE, PT := t#0s);
       //RETURN;
   END_IF;


   // Преобразуем % скорости в отношение
   #rSpeedRatio := #rSpeedPercent / 100.0;

   // Расчёт фактической скорости (м/с)
   #rConveyorSpeed := #rVmax * #rSpeedRatio;

   // Время нахождения бутылки в зоне (мин)
   IF #rConveyorSpeed > 0.0 THEN
       #rHoldTime := #rConveyorLength / #rConveyorSpeed; // В мин
   ELSE
       #rHoldTime := 0.0;
   END_IF;


   IF #bManualMode THEN
       // Ручной режим — берём температуру с панели
       #rTempSetpoint := #rManualTemp;
   ELSE
       // Расчёт температуры по ПЕ
       IF #rHoldTime > 0.0 AND #rPESetpoint > 0.0 THEN
           #rPENeededPerMin := #rPESetpoint / #rHoldTime;
           #rTempSetpoint := #rTref + (LN(#rPENeededPerMin) / LN(#rZParam));


           (*
           #rLogArg := LN(#rPENeededPerMin) / LN(10.0);
           #rTempSetpoint := #rTref + #rLogArg / #rZParam;
           *)
       ELSE
           #rTempSetpoint := #rTref; // по умолчанию
       END_IF;
   END_IF;

   // Проверка пределов
   #bTempValid := TRUE;
   #bAlarmTempHigh := FALSE;
   #bAlarmTempLow := FALSE;


   IF #rTempSetpoint > #rTmax THEN
       #rTempSetpoint := #rTmax;
       #bTempValid := FALSE;
       #bAlarmTempHigh := TRUE;
   ELSIF #rTempSetpoint < #rTmin THEN
       #rTempSetpoint := #rTmin;
       #bTempValid := FALSE;
       #bAlarmTempLow := TRUE;
   END_IF;
END_FUNCTION_BLOCK

FUNCTION_BLOCK "FB_Главный блок конвейера"   // FB12, SCL
{ S7_Optimized_Access := 'TRUE' }
VERSION : 0.1
   VAR_INPUT
      bModePaster : Bool;   // Режим пастеризации
      bModeStiril : Bool;   // Режим сетрилизации
      bModeBanya : Bool;   // Режим Баня
      bAlarmSystem : Bool;   // Общая авария
      bResAlarm : Bool;   // Сброс аварий
      bStartCMD : Bool;   // Подтверждение оператором старта
      bAllZone_Ok : Bool;   // Маркер - все зоны ОК
      bHasPauseKonv : Bool;   // Маркер - пауза конвейера
      tiWaitZone : DInt;   // HMI - мин - Время ожидания выхода на режим
      tiWaitPause : DInt;   // HMI - мин - Время ожидания возврата с паузы
      tiWaitToGoPause : DInt;   // HMI-сек Время задержки для перехода на паузу
      tiWaitToCameGo : DInt;   // HMI- сек Время задержки для возврата в рабочий режим
   END_VAR
   VAR_OUTPUT
      iStep : Int;   // Шаг конвейера
      bKonveyorRun : Bool;   // Разрешение на работу конвейера
      bAlarmToLongPause : Bool;   // Авария по превышения ожидания выхода с паузы
      bAlarmToLongWaitZone_Ok : Bool;   // Авария по превышения ожидания выхода на режим
      bOpenWindOper : Bool;   // вызов окна оператора
   END_VAR
   VAR
      TON_WaitZones : TON_TIME;   // Таймер ожидания перехода в готовность, или в Аварию
      TON_PauseWait : TON_TIME;   // Таймер ожидания возврата с паузы до перехода в аварию
      TON_WaitToGoPaus : TON_TIME;   // Задержка для перехода в паузу
      TON_WaitToComeGo : TON_TIME;   // Задержка для выхода из паузу
      bAlarm_Timer : Bool;   // общий меркер по авариям внутри конве
   END_VAR
   VAR CONSTANT
      S_STOP : Int;   // Шаги
      S_Start_WaitZones : Int := 10;
      S_ConfirmStart : Int := 20;
      S_Working : Int := 30;
      S_Paused : Int := 40;
      S_Sterilization : Int := 50;
      S_Bany : Int := 60;
      S_Alarm : Int := 99;
      ConstMin : DInt := 60000;   // Минуты
      ConstS : DInt := 1000;   // Секунды
   END_VAR
BEGIN

   // Проверяем блок на наличие внешних аварий и наличие разрешения на работу
   #bOpenWindOper := FALSE;


   IF #bAlarmSystem OR #bAlarm_Timer THEN
       #iStep := #S_Alarm;
   ELSIF
       NOT #bModePaster AND NOT #bModeStiril AND NOT #bModeBanya AND NOT (#iStep = #S_Alarm) THEN
       #iStep := #S_STOP;
   END_IF;


   CASE #iStep OF
           //...................................................................................................................................................        
       #S_STOP: // ШАГ - СТОП 0
           //....Сбрасываем таймеры.......
               #TON_WaitToGoPaus(IN := FALSE,
                                 PT := t#0s);
               #TON_WaitToComeGo(IN := FALSE,
                                 PT := t#0s);
               #TON_WaitZones(IN := FALSE,
                              PT := t#0s);
               #TON_PauseWait(IN := FALSE,
                              PT := t#0s);

               #bKonveyorRun := FALSE;


               IF #bModePaster THEN
                   #iStep := #S_Start_WaitZones;
               ELSIF #bModeStiril THEN
                   #iStep := #S_Sterilization;
               ELSIF #bModeBanya THEN
                   #iStep := #S_Start_WaitZones;
               END_IF;

           //...................................................................................................................................................
       #S_Start_WaitZones: // Шаг - Ожидание готовности зон 10
           IF #bAllZone_Ok THEN
               // Если все зоны впорядке сбрасывам таймер ожидания готовности зоны
               #TON_WaitZones(IN := FALSE,
                              PT := #tiWaitZone * #ConstMin);
               #iStep := #S_ConfirmStart;
           ELSE
               #TON_WaitZones(IN := TRUE,
                              PT := #tiWaitZone * #ConstMin);
               IF #TON_WaitZones.Q THEN
                   #bAlarmToLongWaitZone_Ok := TRUE;
                   #iStep := #S_STOP;
               END_IF;
           END_IF;

           //...................................................................................................................................................
       #S_ConfirmStart:    // ШАГ ожидания подтверждения оператора 20
           #bOpenWindOper := #bAllZone_Ok;
           IF #bAllZone_Ok THEN    // Если все зоны готовы то выводим окно оператора и ждем подтверждения
               #bOpenWindOper := TRUE; //Вызов окна оператора
               IF #bStartCMD THEN
                   //#bOpenWindOper := FALSE;
                   #iStep := #S_Working;
               END_IF;
           ELSE
               #iStep := #S_Start_WaitZones;
           END_IF;

           //...................................................................................................................................................            
       #S_Working:         // ШАГ Работа конвейера 30
           IF NOT #bAllZone_Ok THEN
               IF #bHasPauseKonv THEN
                   #TON_WaitToGoPaus(IN := TRUE,
                                     PT := #tiWaitToGoPause * #ConstS);
                   IF #TON_WaitToGoPaus.Q THEN
                       #iStep := #S_Paused;
                   END_IF;
               END_IF;
           ELSE
               #bKonveyorRun := TRUE;

               #TON_WaitToGoPaus(IN := FALSE,
                                 PT := t#0s);
           END_IF;

           //...................................................................................................................................................              
       #S_Paused:          //ШАГ Пауза 40

           #bKonveyorRun := FALSE;

           //Запускаем таймер ожидания предельного времени нахождения в паузе
           #TON_PauseWait(IN := TRUE,
                          PT := #tiWaitPause * #ConstMin);

           // Проверка таймера - если время вышло то АВАРИЯ
           IF #TON_PauseWait.Q THEN
               #bAlarmToLongPause := TRUE;
               #iStep := #S_STOP;
           END_IF;

           // Проверка возврата в рабочий режим - если маркер паузы снят, то возвращаемся в старт
           IF NOT #bHasPauseKonv THEN
               //Сброс таймера Пауза
               #TON_PauseWait(IN := FALSE,
                              PT := t#0s);
               //Старт таймер ожидания возврата к работе
               #TON_WaitToComeGo(IN := TRUE,
                                 PT := #tiWaitToCameGo * #ConstS);

               IF #TON_WaitToComeGo.Q THEN
                   #iStep := #S_Working;
               END_IF;
           ELSE
               #TON_WaitToComeGo(IN := FALSE,
                                 PT := #tiWaitToCameGo * #ConstS);
           END_IF;


           //......................//ШАГ Стерилизиция.............................................................................................................................              
       #S_Sterilization:          

           #bKonveyorRun := FALSE;         //Conveyor - STOP

           //....................................................................................................................................................
           //____________________ Alarm ____________________________


       #S_Alarm:
           #bKonveyorRun := FALSE;
           IF #bResAlarm THEN
               #iStep := #S_STOP;
           END_IF;

   END_CASE;

   // Сброс Аварий
   IF #bResAlarm THEN
       #bAlarmToLongPause := FALSE;
       #bAlarmToLongWaitZone_Ok := FALSE;
   END_IF;
   // Вызов окна подтверждения оператора

   //Флаг АВАРИИ внутренний по таймерам
   #bAlarm_Timer := #bAlarmToLongWaitZone_Ok OR #bAlarmToLongPause;
END_FUNCTION_BLOCK

FUNCTION_BLOCK "FB_Filling_Bac"   // FB17, SCL
{ S7_Optimized_Access := 'TRUE' }
VERSION : 0.1
   VAR_INPUT
      bEnable : Bool;   // Разрешение на работу
      bLevelHigh : Bool;   // Датчик верхнего уровня
      bManualMode : Bool;   // Ручной режим
      bManualOpen : Bool;   // Принудительно открыть клапан в ручном режиме
      "tDelay_O/C" : Time := T#2s;   // Задержка отключения после высокого уровня
   END_VAR
   VAR_OUTPUT
      bValveOpen : Bool;   // Управление клапаном
   END_VAR
   VAR
      bFilling : Bool;   // Внутренний флаг процесса наполнения
      tonDelayOff : TON_TIME;   // Таймер задержки отключения
      tonDelayOn : TON_TIME;   // Таймер задержки включения
   END_VAR
BEGIN

   // Режим ручного управления
   IF #bManualMode THEN
       #bValveOpen := #bManualOpen;

   ELSE
       // Автоматический режим
       IF NOT #bEnable THEN
           // Если нет разрешения — всё выключено
           #bFilling := FALSE;
           #tonDelayOff(IN := FALSE,PT := t#0s);
           #tonDelayOff(IN := FALSE,PT := t#0s);
           #bValveOpen := FALSE;

       ELSE
           // Основная логика управления
           IF NOT #bLevelHigh THEN
               // Запускаем таймер на включение наполнения
               #tonDelayOn(IN := TRUE,
                           PT := #"tDelay_O/C"*1000);

               // Включаем наполнение емкостей
               #bFilling := #tonDelayOn.Q;
           ELSE
               #tonDelayOn(IN := FALSE,
                           PT := #"tDelay_O/C" * 1000);
           END_IF;

           IF #bLevelHigh THEN
               // Запускаем таймер задержки отключения в секундах
               #tonDelayOff(IN := TRUE,
                            PT := #"tDelay_O/C"*1000);

               // Если задержка прошла — отключаем наполнение
               IF #tonDelayOff.Q THEN
                   #bFilling := FALSE;
               END_IF;
           ELSE
               // Если уровень упал — сбрасываем таймер
               #tonDelayOff(IN := FALSE, PT := t#0s);
           END_IF;

           #bValveOpen := #bFilling;
       END_IF;
   END_IF;
END_FUNCTION_BLOCK

FUNCTION_BLOCK "FB_Press_Controll"   // FB18, SCL
{ S7_Optimized_Access := 'TRUE' }
VERSION : 0.1
   VAR_IN_OUT
      DataPress : "tipePress";
   END_VAR
   VAR
      TON_Alarm : TON_TIME;
   END_VAR
BEGIN

   // Если давление ниже уставки в течерии 10 сек - выводим сигнал АВАРИЯ
   // 
   #TON_Alarm(IN := #DataPress.rInPress < #DataPress.rSetpoint, PT := t#10s);

   #DataPress.bAlarm_Press := #TON_Alarm.Q;
END_FUNCTION_BLOCK

FUNCTION_BLOCK "FB_SVETOFOR"   // FB19, SCL
{ S7_Optimized_Access := 'TRUE' }
VERSION : 0.1
   VAR_OUTPUT
      Зеленый : Bool;   // Включение зеленого света
      Желтый : Bool;   // Включение желтого
      Красный : Bool;   // красного
      Пищалка : Bool;
   END_VAR
   VAR
      AlarmPress : Bool;   // Авария по давлению
      bBezz_State : Bool;   // Состояние для выхода
      mAlarm : Bool;   // Сохранение сост АВАРИЯ
      mOpenWind : Bool;   // Сохранение сост Открыто Окно
      mPause : Bool;   // Сохранение сост Пауза
      mSterilFinish : Bool;
   END_VAR
BEGIN
   //Включение зеленого при старте конвейеров
   //
   IF "Разрешение работы конвейера" THEN
       #Зеленый := TRUE;
   ELSIF "bStartWork_Main_TunelPaster" AND NOT "Разрешение работы конвейера" THEN
       #Зеленый := "Time_2s";
   ELSE
       #Зеленый := FALSE;
   END_IF;

   // ___________________________________Упрвавление желтым сигналом________________________
   // 
   #Желтый := FALSE;
   IF "bOpenWindStartConveyor" OR "AlarmPress" OR ("iHMI_Num_StatrPaster" = 40) THEN
       #Желтый := TRUE;
   END_IF;
   IF "bStartWork_Sterilization" AND "bState_Stiril_Zone_OK" THEN
       #Желтый := TRUE;
   ELSIF "bStartWork_Sterilization" AND NOT "bState_Stiril_Zone_OK" THEN
       #Желтый := "Time_2s";
   END_IF;

   //______________________________________Управление карасным сигналом_____________________
   //
   #Красный := FALSE;
   IF "bMain_AlarmSystem" THEN
       #Красный := TRUE;
   END_IF;



   // __________________________________Управление пищалкой-______________________________
   // 
   ///По умолчанию отключаю пищалку
   #bBezz_State := FALSE;
   "RT_Alarm"(CLK:="bMain_AlarmSystem");


   //Условие включения звука при аварии
   IF "RT_Alarm".Q OR #mAlarm THEN
    //   #bBezz_State := TRUE;
       #mAlarm := TRUE;
   END_IF;

   //Условие включения при Вызове вспл окна оператора
   //
   "R_trig_OpenWindOper"(In := "bOpenWindStartConveyor");  //Триггер по открытию окна

   IF NOT "bOpenWindStartConveyor" THEN
       #mOpenWind := FALSE;    //Если окно закрыто - выкл звук

   ELSIF
       "R_trig_OpenWindOper".Q OR #mOpenWind AND NOT "bT_Alarm" THEN
       #mOpenWind := TRUE;

     //  #bBezz_State := "Time_1s";      //Включаем пищалку на цикл по 1 сек

   END_IF;


   // Условие включения при Паузе 
   // 
   "R_trig_Puasa"(In := ("iHMI_Num_StatrPaster" = 40));

   IF "iHMI_Num_StatrPaster" <> 40 THEN    //отключаем пищалку если не в состоянии Пауза
       #mPause := FALSE;
   ELSIF
       "R_trig_Puasa".Q OR #mPause AND NOT "bT_Alarm" THEN
       #mPause := TRUE;

      // #bBezz_State := "Time_1s";  //Включаем пищалку на цикл по 1 сек

   END_IF;

   //Условия для включения при стерилизации

   "RT_Steril_Finish"(CLK:="bHMI_Steril_Fimish");

   IF "RT_Steril_Finish".Q OR #mSterilFinish THEN
       #mSterilFinish := TRUE;
   END_IF;



   //Сбррос пищалки
   //
   IF "bZoomerOff" THEN
       #bBezz_State := FALSE;
       #mPause := FALSE;
       #mOpenWind := FALSE;
       #mAlarm := FALSE;
       #mSterilFinish := FALSE;
       ;
   END_IF;

   //Параметры для выхода на пищалку интенсивность
   IF #mAlarm THEN
       #bBezz_State := TRUE;
   ELSIF #mOpenWind THEN
       #bBezz_State := "Time_1s";
   ELSIF #mPause THEN
       #bBezz_State := "Time_0.5s";
   ELSIF #mSterilFinish THEN
       ;// #bBezz_State := "Time_2s";
   END_IF;

   //Присвоение значения на выход блока
   #Пищалка := #bBezz_State;

   //Вызов окна Операции стирилзации закончена

   "bOpenWindSterilFinish" := #mSterilFinish;
END_FUNCTION_BLOCK

FUNCTION_BLOCK "FB_Zone_Control_Steriliz"   // FB20, SCL
{ S7_Optimized_Access := 'FALSE' }
VERSION : 0.1
   VAR_INPUT
      bNewStart : Bool;   // Обнаружение нового старта, уставка без дельты
      DT_InParamZoneSteril : "Zone_Pararm";
   END_VAR
   VAR_OUTPUT
      ZoneStatusOut : "ZoneStatus";
      bInSetpoint : Bool;
      bOutOfRange : Bool;
      bHasPriority : Bool;
   END_VAR
   VAR
      R_Trig_Start : "R_trig";
      "#bNewStartCLic" : Bool;
      bSetpointReachedOnce : Bool;
   END_VAR
BEGIN
   // --- Сброс флага при необходимости ---
   // 
       //----Отслеживание нажания старта, по верхнему фронту-----
   #R_Trig_Start("In":= #bNewStart,Q => #"#bNewStartCLic");

   IF #"#bNewStartCLic" THEN
       #bSetpointReachedOnce := FALSE;
   END_IF;

   // --- Фиксация первого достижения уставки (точно или ±0.1) ---
   IF NOT #bSetpointReachedOnce AND ABS(#DT_InParamZoneSteril.rTemp - #DT_InParamZoneSteril.rSet) <= 1 THEN
       #bSetpointReachedOnce := TRUE;
   END_IF;

   // --- Расчёт попадания в уставку с учетом асимметричной дельты ---
   IF #bSetpointReachedOnce THEN
       #ZoneStatusOut.bInSetpoint := (#DT_InParamZoneSteril.rTemp >= (#DT_InParamZoneSteril.rSet - #DT_InParamZoneSteril.rDeltaDown)) AND
       (#DT_InParamZoneSteril.rTemp <= (#DT_InParamZoneSteril.rSet + #DT_InParamZoneSteril.rDeltaUP));
   ELSE
       // До первого достижения — строгое приближение (или узкая дельта)
       #ZoneStatusOut.bInSetpoint := ABS(#DT_InParamZoneSteril.rTemp - #DT_InParamZoneSteril.rSet) <= 1;
   END_IF;

   //Контроль зоны выхода из уставок значительно, греем снова до уставки до разрешения на старт

   IF (#DT_InParamZoneSteril.rTemp < (#DT_InParamZoneSteril.rSet - #DT_InParamZoneSteril.rDeltaDown)) OR
       (#DT_InParamZoneSteril.rTemp > (#DT_InParamZoneSteril.rSet + #DT_InParamZoneSteril.rDeltaUP)) THEN
       #bSetpointReachedOnce := FALSE;
   END_IF;


   // --- Остальные сигналы ---
   #ZoneStatusOut.bOutOfRange := NOT #ZoneStatusOut.bInSetpoint;
   #ZoneStatusOut.bHasPriority := #DT_InParamZoneSteril.bPriority;

   // Зеркалируем, если нужно
   #bInSetpoint := #ZoneStatusOut.bInSetpoint;
   #bOutOfRange := #ZoneStatusOut.bOutOfRange;
   #bHasPriority := #ZoneStatusOut.bHasPriority;
END_FUNCTION_BLOCK

FUNCTION_BLOCK "FB_Steril_Timer"   // FB22, SCL
{ S7_Optimized_Access := 'TRUE' }
VERSION : 0.1
   VAR_INPUT
      En_1 : Bool;   // Разрешение работы блока
      Start : Bool;   // Старт / Пауза
      SetTimeMin : Int;   // Уставка в минутах (задаётся с HMI)
   END_VAR
   VAR_OUTPUT
      RemainingMin : Int;   // Оставшиеся минуты
      RemainingSec : Int;   // Оставшиеся секунды
      TimeIsUp : Bool;   // Флаг конца времени
   END_VAR
   VAR
      TotalSec : DInt;   // Полное время в сек
      RemSec : DInt;   // Отсаток в сек
      bStartPrev : Bool;   // Для фронта
      bSecPulse : Bool;   // Секунда имп
      ton1 : TON_TIME;   // отсчет 1 сек
   END_VAR
BEGIN
   // ---------------------------------------------------------
   // Инициализация при EN = FALSE
   // ---------------------------------------------------------
   IF NOT #En_1 THEN
       #TotalSec := #SetTimeMin * 60;  // Пересчёт уставки в секунды
       #RemSec := #TotalSec;
       #RemainingMin := #SetTimeMin;
       #RemainingSec := 0;
       #TimeIsUp := FALSE;
       #ton1(IN := FALSE, PT := t#0s);
       RETURN;
   END_IF;

   // ---------------------------------------------------------
   // Генерация секундного импульса через TON (1 сек)
   // ---------------------------------------------------------
   #ton1(IN := #Start,
         PT := T#1S);

   IF #ton1.Q THEN
       #bSecPulse := TRUE;
       #ton1(IN := FALSE, PT := t#0s); // перезапуск таймера
   ELSE
       #bSecPulse := FALSE;
   END_IF;

   // ---------------------------------------------------------
   // Основная логика обратного отсчёта
   // ---------------------------------------------------------
   IF #Start AND (#RemSec > 0) THEN
       IF #bSecPulse THEN
           #RemSec := #RemSec - 1;
       END_IF;
   END_IF;

   // ---------------------------------------------------------
   // Если время вышло
   // ---------------------------------------------------------
   IF #RemSec <= 0 THEN
       #RemSec := 0;
       #TimeIsUp := TRUE;
   ELSE
       #TimeIsUp := FALSE;
   END_IF;

   // ---------------------------------------------------------
   // Преобразование остатка в минуты и секунды
   // ---------------------------------------------------------
   #RemainingMin := #RemSec / 60;
   #RemainingSec := #RemSec MOD 60;
END_FUNCTION_BLOCK

FUNCTION_BLOCK "FB_CheckZoneStatus"   // FB23, SCL
{ S7_Optimized_Access := 'FALSE' }
VERSION : 0.1
   VAR_OUTPUT
      bAllZones_Redy : Bool;   // Выход состояния всех зон ОК
      bPriority_Stop : Bool;   // Выход 1 - если есть метка остановки конвейера
      iZonesNumberFail : Int;   // ВЫход с Номером зоны
   END_VAR
   VAR
      aZoneS_Status : Array[1..10] of "ZoneStatus";   // Массив с данными по всем зонам
      i : Int;
      AllZone_Ok : Bool;   // Состояние всех зон ОК
      HaveStopPriority : Bool;   // В зоне есть метка для остановки конвейера
      iNumber : Int;   // Номер зоны, где отклонение температуры
   END_VAR
BEGIN

   //Что бы не контролировал готовность зоны 4 ее не надо контролировать
   //"ЗОНЫ_Параметры".Zone_4.bOUT_ZoneStatus.bInSetpoint := TRUE;
   //-------------------------------------------------------------------------------------------//
   //
           // ----Сбор данных по всем зонам в массив для обработки-----

           #aZoneS_Status[4] := "Зоны_Баня_Парам"."Banya_Zona-4".bOUT_ZoneStatus;
           #aZoneS_Status[5] := "Зоны_Баня_Парам"."Banya_Zona-5".bOUT_ZoneStatus;
           #aZoneS_Status[6] := "Зоны_Баня_Парам"."Banya_Zona-6".bOUT_ZoneStatus;



           //Сброс маркеров по умолчанию----
   #AllZone_Ok := TRUE;    
   #HaveStopPriority := FALSE;
   #iNumber := 0;
              // ----Цикл для перебора всех зон значение выставить по количеству зон----
   FOR #i := 4 TO 6 DO
      (* 
       IF (#i = 5 OR #i = 6) THEN  //Пропускаем статусы зон
           CONTINUE;
       END_IF;
       *)
       IF NOT #aZoneS_Status[#i].bInSetpoint THEN
           #AllZone_Ok := FALSE;
           #iNumber := #i;
           IF #aZoneS_Status[#i].bHasPriority THEN
               #HaveStopPriority := TRUE;
           END_IF;
       END_IF;
   END_FOR;

   /// Присвоение переменных к выходам
   #bAllZones_Redy := #AllZone_Ok;
   #bPriority_Stop := #HaveStopPriority;
   #iZonesNumberFail := #iNumber;
END_FUNCTION_BLOCK

FUNCTION_BLOCK "Test_Beep"   // FB24, SCL
{ S7_Optimized_Access := 'TRUE' }
VERSION : 0.1
   VAR
      BzzzState : Bool;
      mOpWind : Bool;
      mPause : Bool;
      mAlarm : Bool;
   END_VAR
BEGIN
   #BzzzState := FALSE;
   //Условие включения звука при аварии
   IF "bT_Alarm" OR #mAlarm THEN
      // #BzzzState := TRUE;
       #mAlarm := TRUE;
   END_IF;

   //Условие включения при Вызове вспл окна оператора
   //
   "R_TRIG_TestOpenWind"(CLK:="bTOpenWind");
   IF NOT "bTOpenWind" THEN
       #mOpWind := FALSE;

   ELSIF
       "R_TRIG_TestOpenWind".Q OR #mOpWind AND NOT "bT_Alarm" THEN
      // #BzzzState := "Time_0.5s";
       #mOpWind := TRUE;
   END_IF;



   // Условие включения при Паузе 
   // 
   "R_TRIG_TestPause"(CLK:=("iTestPause" = 40));


   IF "iTestPause" <> 40 THEN
       #mPause := FALSE;
   ELSIF
       "R_TRIG_TestPause".Q OR #mPause AND NOT "bT_Alarm" THEN
       //#BzzzState := "Time_0.2s";
       #mPause := TRUE;
   END_IF;
   ;

   //Сбррос пищалки
   //
   IF "bTZoomOff" THEN
       #BzzzState := FALSE;
       #mPause := FALSE;
       #mOpWind := FALSE;
       #mAlarm := FALSE;
       ;
   END_IF;

   IF #mAlarm THEN
       #BzzzState := TRUE;
   ELSIF #mOpWind THEN
       #BzzzState := "Time_1s";
   ELSIF #mPause THEN
       #BzzzState := "Time_0.5s";
   END_IF;
END_FUNCTION_BLOCK

FUNCTION_BLOCK "FB_Mode_STIRIL"   // FB25, SCL
{ S7_Optimized_Access := 'TRUE' }
VERSION : 0.1
   VAR_INPUT
      bEn_Mode : Bool;   // разрешение на работу
   END_VAR
BEGIN
   IF NOT #bEn_Mode THEN
       RETURN;
   END_IF;

   IF #bEn_Mode THEN
       //Открываем калпана запорные
       "FVs_o/p".FV_5.bOpenCmd := TRUE;    //Клапан пара
       "FVs_o/p".FV_1.bOpenCmd := TRUE;    //Клапан Стерилизации

       //Открываем клапана регулирующие
       "FVs_Regul".FV_Regul_1."bAutoOpen/Close" := TRUE;
       "FVs_Regul".FV_Regul_2."bAutoOpen/Close" := TRUE;
       "FVs_Regul".FV_Regul_3."bAutoOpen/Close" := TRUE;
       "FVs_Regul".FV_Regul_4."bAutoOpen/Close" := TRUE;
       "FVs_Regul".FV_Regul_5."bAutoOpen/Close" := TRUE;
       "FVs_Regul".FV_Regul_6."bAutoOpen/Close" := TRUE;
       "FVs_Regul".FV_Regul_7."bAutoOpen/Close" := FALSE;
       "FVs_Regul".FV_Regul_8."bAutoOpen/Close" := TRUE;
       "FVs_Regul".FV_Regul_9."bAutoOpen/Close" := TRUE;
       "FVs_Regul".FV_Regul_10."bAutoOpen/Close" := TRUE;
       "FVs_Regul".FV_Regul_11."bAutoOpen/Close" := TRUE;
       "FVs_Regul".FV_Regul_12."bAutoOpen/Close" := TRUE;


       //Передача уставки для пид регуляторов
       //
       "Param_PID".k_PID_Zona1.Set := "Зоны_Стерилизации_Парам"."Steril_Zona-1".rSet;
       "Param_PID".k_PID_Zona2.Set := "Зоны_Стерилизации_Парам"."Steril_Zona-2".rSet;
       "Param_PID".k_PID_Zona3.Set := "Зоны_Стерилизации_Парам"."Steril_Zona-3".rSet;
       "Param_PID".k_PID_Zona4.Set := "Зоны_Стерилизации_Парам"."Steril_Zona-4".rSet;
       "Param_PID".k_PID_Zona5.Set := "Зоны_Стерилизации_Парам"."Steril_Zona-5".rSet;
       "Param_PID".k_PID_Zona6.Set := "Зоны_Стерилизации_Парам"."Steril_Zona-6".rSet;


       ;


       //Старт насосов
       //
       "Pumps".Pump_1.bAutoMode_Work := TRUE;
       "Pumps".Pump_2.bAutoMode_Work := TRUE;
       "Pumps".Pump_3.bAutoMode_Work := TRUE;
       "Pumps".Pump_4.bAutoMode_Work := TRUE;
       "Pumps".Pump_5.bAutoMode_Work := TRUE;
       "Pumps".Pump_6.bAutoMode_Work := TRUE;
       "Pumps".Pump_7.bAutoMode_Work := TRUE;
       "Pumps".Pump_8.bAutoMode_Work := TRUE;
       "Pumps".Pump_9.bAutoMode_Work := TRUE;
       "Pumps".Pump_10.bAutoMode_Work := TRUE;




   END_IF;
END_FUNCTION_BLOCK

FUNCTION_BLOCK "FB_Mode_Paster"   // FB26, SCL
{ S7_Optimized_Access := 'TRUE' }
VERSION : 0.1
   VAR_INPUT
      bEn_Mode : Bool;   // разрешение на работу
      bSafetyMode : Bool;   // Режим защиты от перепастеризации
      bOn_Safety : Bool;   // Сигнал на переход в режим защиты
      bResetSafety : Bool;   // Сигнал сброса режима защиты
   END_VAR
BEGIN
   IF NOT #bEn_Mode THEN
       RETURN;
   END_IF;

           //Старт насосов
           //
           "Pumps".Pump_1.bAutoMode_Work := TRUE;
           "Pumps".Pump_2.bAutoMode_Work := TRUE;
           "Pumps".Pump_3.bAutoMode_Work := TRUE;
           "Pumps".Pump_4.bAutoMode_Work := TRUE;
           "Pumps".Pump_5.bAutoMode_Work := TRUE;
           "Pumps".Pump_6.bAutoMode_Work := TRUE;
           "Pumps".Pump_7.bAutoMode_Work := TRUE;
           "Pumps".Pump_8.bAutoMode_Work := TRUE;
           "Pumps".Pump_9.bAutoMode_Work := TRUE;
           "Pumps".Pump_10.bAutoMode_Work := TRUE;

       //Открываем калпана запорные

       "FVs_o/p".FV_5.bOpenCmd := NOT #bOn_Safety AND #bSafetyMode;    //Клапан пара работает если нет режима защиты от перепастеризации
      // "FVs_o/p".FV_1.bOpenCmd := FALSE;    //Клапан Стерилизации

       //==================================================================================
      //============== Работа системы в режиме ПАСТЕРИЗАЦИИ ================
      //====================================================================

       //Открываем клапана регулирующие
       "FVs_Regul".FV_Regul_1."bAutoOpen/Close" := TRUE;
       "FVs_Regul".FV_Regul_2."bAutoOpen/Close" := TRUE;
       "FVs_Regul".FV_Regul_3."bAutoOpen/Close" := TRUE;
       "FVs_Regul".FV_Regul_4."bAutoOpen/Close" := TRUE;
       "FVs_Regul".FV_Regul_5."bAutoOpen/Close" := TRUE;
       "FVs_Regul".FV_Regul_6."bAutoOpen/Close" := TRUE;
       "FVs_Regul".FV_Regul_7."bAutoOpen/Close" := TRUE;

       //Клапана защиты от перепастеризации - закрыты
       "FVs_Regul".FV_Regul_8."bAutoOpen/Close" := FALSE;
       "FVs_Regul".FV_Regul_9."bAutoOpen/Close" := FALSE;
       "FVs_Regul".FV_Regul_10."bAutoOpen/Close" := FALSE;
       "FVs_Regul".FV_Regul_11."bAutoOpen/Close" := FALSE;
       "FVs_Regul".FV_Regul_12."bAutoOpen/Close" := FALSE;

       //Передача уставки для пид регуляторов
       //
       "Param_PID".k_PID_Zona1.Set := "ЗОНЫ_Параметры".Zone_1.rSet;
       "Param_PID".k_PID_Zona2.Set := "ЗОНЫ_Параметры".Zone_2.rSet;
       "Param_PID".k_PID_Zona3.Set := "ЗОНЫ_Параметры".Zone_3.rSet;
       "Param_PID".k_PID_Zona4.Set := "ЗОНЫ_Параметры".Zone_4.rSet;
       "Param_PID".k_PID_Zona5.Set := "ЗОНЫ_Параметры".Zone_5.rSet;
       "Param_PID".k_PID_Zona6.Set := "ЗОНЫ_Параметры".Zone_6.rSet;
       "Param_PID".k_PID_Zona10.Set := "ЗОНЫ_Параметры".Zone_10.rSet;

       //==================================================================================
       //============== Работа системы в режиме защиты от Перепастеризации ================
       //==================================================================================

       IF #bSafetyMode AND #bOn_Safety THEN
           //Клапана нагрева - закрывваем
           "FVs_Regul".FV_Regul_1."bAutoOpen/Close" := FALSE;
           "FVs_Regul".FV_Regul_2."bAutoOpen/Close" := FALSE;
           "FVs_Regul".FV_Regul_3."bAutoOpen/Close" := FALSE;
           "FVs_Regul".FV_Regul_4."bAutoOpen/Close" := FALSE;
           "FVs_Regul".FV_Regul_5."bAutoOpen/Close" := FALSE;
           "FVs_Regul".FV_Regul_6."bAutoOpen/Close" := FALSE;
           "FVs_Regul".FV_Regul_7."bAutoOpen/Close" := FALSE;

           //Клапана защиты от перепастеризации - открываем
           "FVs_Regul".FV_Regul_8."bAutoOpen/Close" := TRUE;
           "FVs_Regul".FV_Regul_9."bAutoOpen/Close" := TRUE;
           "FVs_Regul".FV_Regul_10."bAutoOpen/Close" := TRUE;
           "FVs_Regul".FV_Regul_11."bAutoOpen/Close" := TRUE;
           "FVs_Regul".FV_Regul_12."bAutoOpen/Close" := TRUE;

           //Передача уставки для пид регуляторов
           //

           "Param_PID".k_PID_Zona3.Set := "Param_PID".k_PID_Zona3_Охл.Set;
           "Param_PID".k_PID_Zona4.Set := "Param_PID".k_PID_Zona4_Охл.Set;
           "Param_PID".k_PID_Zona5.Set := "Param_PID".k_PID_Zona5_Охл.Set;
           "Param_PID".k_PID_Zona6.Set := "Param_PID".k_PID_Zona6_Охл.Set;
           "Param_PID".k_PID_Zona10.Set := "Param_PID".k_PID_Zona7_Охл.Set;

       END_IF;
END_FUNCTION_BLOCK

FUNCTION_BLOCK "Насос химии"   // FB27, SCL
{ S7_Optimized_Access := 'TRUE' }
VERSION : 0.1
   VAR_INPUT
      bFlip_En : Bool;
      Time_Flip : DInt := 1;
      Time_Pause : DInt := 10;
   END_VAR
   VAR_OUTPUT
      bWorkPump : Bool;
   END_VAR
   VAR
      iflip_step : Int;
      TON_Flip : TON_TIME;
      TON_Pause : TON_TIME;
      tTime_Flim_sec : DInt;
      tTime_Flim_Pause : DInt;
   END_VAR
BEGIN
   #tTime_Flim_sec := #Time_Flip * 1000;
   #tTime_Flim_Pause := #Time_Pause * 1000;

   IF #bFlip_En THEN
       CASE #iflip_step OF

           0:
               //Стоп флип
               #bWorkPump := FALSE;

               #TON_Pause(IN := TRUE,
                          PT := #tTime_Flim_Pause);
               IF #TON_Pause.Q THEN
                   #iflip_step := 1;
               END_IF;

           1:  //Флип клапан 4

               #TON_Flip.TON(IN := true,
                             PT := #tTime_Flim_sec);   //Time for next step

               #bWorkPump := TRUE;

               #TON_Pause(IN := FALSE,
                          PT := t#0s);

               //Переход на следующий шаг по завершению таймера
               IF #TON_Flip.Q THEN
                   #iflip_step := 0;
                   #TON_Flip.TON(IN := FALSE,
                                 PT := t#0s);
               END_IF;


       END_CASE;

   ELSE
       #bWorkPump := FALSE;

       #TON_Pause(IN := FALSE,
                  PT := t#0s);
       #iflip_step := 0;
   END_IF;
END_FUNCTION_BLOCK

FUNCTION_BLOCK "FB_Mode_Bany"   // FB28, SCL
{ S7_Optimized_Access := 'TRUE' }
VERSION : 0.1
   VAR_INPUT
      bEn_Bany : Bool;
   END_VAR
BEGIN
   IF NOT #bEn_Bany THEN
       RETURN;
   END_IF;

   IF #bEn_Bany THEN
       //Открываем калпана запорные
       "FVs_o/p".FV_5.bOpenCmd := TRUE;    //Клапан пара
       //"FVs_o/p".FV_1.bOpenCmd := TRUE;    //Клапан Стерилизации

       //Открываем клапана регулирующие
       "FVs_Regul".FV_Regul_1."bAutoOpen/Close" := FALSE;
       "FVs_Regul".FV_Regul_2."bAutoOpen/Close" := FALSE;
       "FVs_Regul".FV_Regul_3."bAutoOpen/Close" := FALSE;
       //__________________________________________________________
       "FVs_Regul".FV_Regul_4."bAutoOpen/Close" := TRUE;
       "FVs_Regul".FV_Regul_5."bAutoOpen/Close" := TRUE;
       "FVs_Regul".FV_Regul_6."bAutoOpen/Close" := TRUE;
       //__________________________________________________________
       "FVs_Regul".FV_Regul_7."bAutoOpen/Close" := FALSE;
       "FVs_Regul".FV_Regul_8."bAutoOpen/Close" := FALSE;
       "FVs_Regul".FV_Regul_9."bAutoOpen/Close" := FALSE;
       "FVs_Regul".FV_Regul_10."bAutoOpen/Close" := FALSE;
       "FVs_Regul".FV_Regul_11."bAutoOpen/Close" := FALSE;
       "FVs_Regul".FV_Regul_12."bAutoOpen/Close" := FALSE;


       //Передача уставки для пид регуляторов
       //
       "Param_PID".k_PID_Zona4.Set := "Зоны_Баня_Парам"."Banya_Zona-4".rSet;
       "Param_PID".k_PID_Zona5.Set := "Зоны_Баня_Парам"."Banya_Zona-5".rSet;
       "Param_PID".k_PID_Zona6.Set := "Зоны_Баня_Парам"."Banya_Zona-6".rSet;

       ;


       //Старт насосов
       //
       "Pumps".Pump_1.bAutoMode_Work := FALSE;
       "Pumps".Pump_2.bAutoMode_Work := FALSE;
       "Pumps".Pump_3.bAutoMode_Work := FALSE;
       //__________________________________________________________
       "Pumps".Pump_4.bAutoMode_Work := TRUE;
       "Pumps".Pump_5.bAutoMode_Work := TRUE;
       "Pumps".Pump_6.bAutoMode_Work := TRUE;
       //__________________________________________________________
       "Pumps".Pump_7.bAutoMode_Work := FALSE;
       "Pumps".Pump_8.bAutoMode_Work := FALSE;
       "Pumps".Pump_9.bAutoMode_Work := FALSE;
       "Pumps".Pump_10.bAutoMode_Work := FALSE;



   END_IF;
END_FUNCTION_BLOCK

FUNCTION_BLOCK "FB_Защита от Перепастеризации"   // FB29, SCL
{ S7_Optimized_Access := 'TRUE' }
VERSION : 0.1
   VAR_INPUT
      bEn : Bool;
      bAlarmSignal : Bool;   // Сигнал перехода в защиту от перепастеризации
      TimeWaitingToSafety : DInt;   // СЕК, Время ожидания при появлении сигнала перехода к защите
      bResetSafetyMode : Bool;   // Сигнал сброса режиа защиты от перепастеризации
   END_VAR
   VAR_OUTPUT
      bOutSafetyMode : Bool;
   END_VAR
   VAR
      TON_Waiting : TON_TIME;   // Таймер ожидания
      Time_SEC : DInt;
   END_VAR
BEGIN
   //Контроль разрешения на работу блока
   IF NOT #bEn THEN
       RETURN;
   END_IF;

   //===========__Задаем время ожидания перехода в режим защиты от перепастеризации в СЕК___==============================

   #Time_SEC := #TimeWaitingToSafety * 1000;

   #TON_Waiting (IN:=#bAlarmSignal,
                 PT:=#Time_SEC);
   //____________________Переход в режим защиты при отработке таймера___________________________

   IF #TON_Waiting.Q THEN
       #bOutSafetyMode := TRUE;
   END_IF;

   //____________________Сброс режима защиты только по нажатию клавиши ресет___________________________
   //
   IF #bResetSafetyMode THEN
       #bOutSafetyMode := FALSE;
   END_IF;
END_FUNCTION_BLOCK